// ---- Devices/Basic/FB_DeviceReal.TcPOU
(*
	Basic device with extended interface:
	nControl BYTE: From TwinCAT >>> To Unity
	nStatus BYTE: FROM Unity >>> TO TwinCAT	
	fControlData REAL: From TwinCAT >>> To Unity
	fStatusData REAL: FROM Unity >>> TO TwinCAT	
*)
FUNCTION_BLOCK FB_DeviceReal EXTENDS FB_LinkDataReal
VAR_INPUT		
	nControl  			: BYTE;
	fControlData  		: REAL;
END_VAR

VAR_OUTPUT
	nStatus  			: BYTE;
	fStatusData  		: REAL;
END_VAR

SUPER^();
Control := nControl;
ControlData := fControlData;
nStatus := Status;
fStatusData := StatusData;

END_FUNCTION_BLOCK

// ---- Common/Links/FB_LinkDataReal.TcPOU
(*
	Link component with additional interface:
	Control BYTE: From TwinCAT >>> To Unity	(Default)
	Status BYTE: FROM Unity >>> TO TwinCAT	(Default)
	ControlData REAL: From TwinCAT >>> To Unity		
	StatusData REAL: FROM Unity >>> TO TwinCAT		
*)
FUNCTION_BLOCK FB_LinkDataReal EXTENDS FB_LinkDevice
VAR	
	{attribute 'simulation_interface'}
	ControlData			AT %Q* : REAL;
	{attribute 'simulation_interface'}
	StatusData			AT %I* : REAL;
END_VAR

SUPER^();

METHOD INTERNAL GetLinkControlData : REAL
GetLinkControlData := ControlData;
END_METHOD

METHOD INTERNAL SetLinkStatusData : BOOL
VAR_INPUT
	fStatusData : REAL;
END_VAR
StatusData := fStatusData;
END_METHOD

END_FUNCTION_BLOCK

// ---- Tests/Devices/FB_Drive_Test.TcPOU
FUNCTION_BLOCK FB_Drive_Test EXTENDS TcUnit.FB_TestSuite
VAR
	_fbDrive 			: FB_Drive;
	_nExpectedByte 		: BYTE;
	_nResultByte 		: BYTE;
	_fExpectedReal 		: REAL;
	_fResultReal 		: REAL;
END_VAR

TEST('Set nControl');
_nExpectedByte := 255;
_fbDrive.nControl := _nExpectedByte;
_fbDrive();
_nResultByte := _fbDrive.GetControl();

AssertEquals(Expected := _nExpectedByte,
             Actual := _nResultByte,
             Message := 'Value is not correct');	
TEST_FINISHED();

TEST('Get nStatus');
_nExpectedByte := 255;
_fbDrive.SetStatus(_nExpectedByte);
_fbDrive();
_nResultByte := _fbDrive.nStatus;

AssertEquals(Expected := _nExpectedByte,
             Actual := _nResultByte,
             Message := 'Value is not correct');	
TEST_FINISHED();

TEST('Set fTargetValue_1');
_fExpectedReal := 1000;
_fbDrive.fTargetValue := _fExpectedReal;
_fbDrive();
_fResultReal := _fbDrive.GetLinkControlData();

AssertEquals(Expected := _fExpectedReal,
             Actual := _fResultReal,
             Message := 'Value is not correct');	
TEST_FINISHED();

TEST('Set fTargetValue_2');
_fExpectedReal := -1000;
_fbDrive.fTargetValue := _fExpectedReal;
_fbDrive();
_fResultReal := _fbDrive.GetLinkControlData();

AssertEquals(Expected := _fExpectedReal,
             Actual := _fResultReal,
             Message := 'Value is not correct');	
TEST_FINISHED();

TEST('Get fActualValue_1');
_fExpectedReal := 1000;
_fbDrive.SetLinkStatusData(_fExpectedReal);
_fbDrive();
_fResultReal := _fbDrive.fActualValue;

AssertEquals(Expected := _fExpectedReal,
             Actual := _fResultReal,
             Message := 'Value is not correct');	
TEST_FINISHED();

TEST('Get fActualValue_2');
_fExpectedReal := -1000;
_fbDrive.SetLinkStatusData(_fExpectedReal);
_fbDrive();
_fResultReal := _fbDrive.fActualValue;

AssertEquals(Expected := _fExpectedReal,
             Actual := _fResultReal,
             Message := 'Value is not correct');	
TEST_FINISHED();

END_FUNCTION_BLOCK

// ---- Devices/Basic/FB_Drive.TcPOU
(*
	Basic drive interface:
	nControl BYTE: From TwinCAT >>> To Unity
	nStatus BYTE: FROM Unity >>> TO TwinCAT	
	fTargetValue REAL: From TwinCAT >>> To Unity
	fActualValue REAL: FROM Unity >>> TO TwinCAT	
*)
FUNCTION_BLOCK FB_Drive EXTENDS FB_LinkDataREAL
VAR_INPUT
	nControl  		: BYTE;
	fTargetValue 	: REAL; //Target value to drive
END_VAR

VAR_OUTPUT
	nStatus  		: BYTE;
	fActualValue 	: REAL; //Actual value from drive
END_VAR

SUPER^();
Control := nControl;
ControlData := fTargetValue;
nStatus := Status;
fActualValue := StatusData;

END_FUNCTION_BLOCK

// ---- Tests/Devices/FB_Lamp_Test.TcPOU
FUNCTION_BLOCK FB_Lamp_Test EXTENDS TcUnit.FB_TestSuite
VAR
	_fbLamp : FB_Lamp;
	_nExpected : BYTE;
	_nResult : BYTE;
	_bExpected : BOOL;
	_bResult : BOOL;
END_VAR

TEST('Set bEnable TRUE');			 
_fbLamp.bEnable := TRUE; 
_fbLamp();
_nExpected := 1;
_nResult := _fbLamp.GetControl();
AssertEquals(Expected := _nExpected,
             Actual := _nResult,
             Message := 'Control value is not correct');	 
TEST_FINISHED();

TEST('Set bEnable FALSE');			 
_fbLamp.bEnable := FALSE; 
_fbLamp();
_nExpected := 0;
_nResult := _fbLamp.GetControl();
AssertEquals(Expected := _nExpected,
             Actual := _nResult,
             Message := 'Control value is not correct');	 
TEST_FINISHED();

END_FUNCTION_BLOCK

// ---- Devices/Basic/FB_Lamp.TcPOU
(*
	Default Lamp device
*)
FUNCTION_BLOCK FB_Lamp EXTENDS FB_LinkDevice 
VAR_INPUT
	bEnable		: BOOL; //0-Lamp OFF, 1 - Lamp ON
END_VAR

SUPER^();
Control.0 := bEnable;

END_FUNCTION_BLOCK

// ---- Tests/Devices/FB_Reader_Test.TcPOU
FUNCTION_BLOCK FB_Reader_Test EXTENDS TcUnit.FB_TestSuite
VAR
	_fbDevice 		: FB_Reader;
	_nExpected 		: LWORD;
	_nResult 		: LWORD;
	_nValue 		: LWORD := 16#FFAABBCC;
END_VAR

TEST('Set nControl');
_nExpected := 255;
_fbDevice.nControl := 255;
_fbDevice();
_nResult := _fbDevice.GetControl();

AssertEquals(Expected := _nExpected,
             Actual := _nResult,
             Message := 'Value is not correct');	
TEST_FINISHED();

TEST('Set nCommand');
_nExpected := _nValue;
_fbDevice.nCommand := _nExpected;
_fbDevice();
_nResult := _fbDevice.GetLinkControlData();

AssertEquals(Expected := _nExpected,
             Actual := _nResult,
             Message := 'Value is not correct');	
TEST_FINISHED();

TEST('Get nStatus');
_nExpected := 255;
_fbDevice.SetStatus(255);
_fbDevice();
_nResult := _fbDevice.nStatus;

AssertEquals(Expected := _nExpected,
             Actual := _nResult,
             Message := 'Value is not correct');	
TEST_FINISHED();

TEST('Get nResult');
_nExpected := _nValue;
_fbDevice.SetLinkStatusData(_nExpected);
_fbDevice();
_nResult := _fbDevice.nResult;

AssertEquals(Expected := _nExpected,
             Actual := _nResult,
             Message := 'Value is not correct');	
TEST_FINISHED();

END_FUNCTION_BLOCK

// ---- Devices/Basic/FB_Reader.TcPOU
(*
	Default reader device	
*)
FUNCTION_BLOCK FB_Reader EXTENDS FB_LinkDataLWORD
VAR_INPUT
	nControl  		: BYTE;
	nCommand 		: ULINT; //Command ID
END_VAR

VAR_OUTPUT
	nStatus  		: BYTE;
	nResult			: ULINT; //Result Data
END_VAR

SUPER^();
Control := nControl;
ControlData := ULINT_TO_LWORD(nCommand);
nStatus := Status;
nResult := LWORD_TO_ULINT(StatusData);

END_FUNCTION_BLOCK

// ---- Tests/Devices/FB_SensorAnalog_Test.TcPOU
FUNCTION_BLOCK FB_SensorAnalog_Test EXTENDS TcUnit.FB_TestSuite
VAR
	_fbSensorAnalog 	: FB_SensorAnalog;
	_nExpectedByte 		: BYTE;
	_nResultByte 		: BYTE;
	_nExpectedUInt 		: UINT;
	_nResultUInt 		: UINT;
	_fExpectedReal 		: REAL;
	_fResultReal 		: REAL;
END_VAR

TEST('Set nControl');
_nExpectedByte := 255;
_fbSensorAnalog.nControl := _nExpectedByte;
_fbSensorAnalog();
_nResultByte := _fbSensorAnalog.GetControl();

AssertEquals(Expected := _nExpectedByte,
             Actual := _nResultByte,
             Message := 'Value is not correct');	
TEST_FINISHED();

TEST('Get nStatus');
_nExpectedByte := 255;
_fbSensorAnalog.SetStatus(_nExpectedByte);
_fbSensorAnalog();
_nResultByte := _fbSensorAnalog.nStatus;

AssertEquals(Expected := _nExpectedByte,
             Actual := _nResultByte,
             Message := 'Value is not correct');	
TEST_FINISHED();


TEST('Get fValue');
_fExpectedReal := 50;
_nExpectedUInt := 16#8000;
_fbSensorAnalog.SetLinkStatusData(_fExpectedReal);
_fbSensorAnalog();
_fResultReal := _fbSensorAnalog.fValue;
_nResultUInt := _fbSensorAnalog.nValue;

AssertEquals(Expected := _fExpectedReal,
             Actual := _fResultReal,
             Message := 'fValue is not correct');	
AssertEquals(Expected := _nExpectedUInt,
             Actual := _nResultUInt,
             Message := 'nValue is not correct');
TEST_FINISHED();

END_FUNCTION_BLOCK

// ---- Devices/Basic/FB_SensorAnalog.TcPOU
(*
	Default analog sensor device. 
	The stConfig structure is used to configure the scaling factor for transforming values into real-world units.
*)
FUNCTION_BLOCK FB_SensorAnalog EXTENDS FB_LinkDataReal 
VAR_INPUT
	nControl  		: BYTE;
	stConfig		: ST_ScaleConfig;
END_VAR

VAR_OUTPUT	
	nStatus  		: BYTE;
	nValue			: UINT;
	fValue			: REAL;
END_VAR

SUPER^();
Control := nControl;
fValue := StatusData;
nValue := LREAL_TO_UINT(F_ScaleLREAL(fValue, stConfig.fInputMin, stConfig.fInputMax, stConfig.fOutputMin, stConfig.fOutputMax));
nStatus := Status;

END_FUNCTION_BLOCK

// ---- Tests/Devices/FB_SensorBinary_Test.TcPOU
FUNCTION_BLOCK FB_SensorBinary_Test EXTENDS TcUnit.FB_TestSuite
VAR
	_fbSensorBinary 	: FB_SensorBinary;
	_nExpected 			: BYTE;
	_nResult 			: BYTE;
	_bExpected 			: BOOL;
	_bResult 			: BOOL;
END_VAR

TEST('Get bValue FALSE');
_fbSensorBinary.SetStatus(0);
_fbSensorBinary();
_bExpected := FALSE;
_bResult := _fbSensorBinary.bValue;

AssertEquals(Expected := _bExpected,
             Actual := _bResult,
             Message := 'Value is not correct');	
TEST_FINISHED();

TEST('Get bValue TRUE');	
_fbSensorBinary.SetStatus(1);
_fbSensorBinary();
_bExpected := 1;
_bResult := _fbSensorBinary.bValue;
AssertEquals(Expected := _bExpected,
             Actual := _bResult,
             Message := 'Control value is not correct');	 
TEST_FINISHED();

END_FUNCTION_BLOCK

// ---- Devices/Basic/FB_SensorBinary.TcPOU
(*
	Default binary sensor device.
*)
FUNCTION_BLOCK FB_SensorBinary EXTENDS FB_LinkDevice 
VAR_OUTPUT
	bValue		: BOOL; 
END_VAR

SUPER^();
bValue := Status.0;

END_FUNCTION_BLOCK

// ---- Tests/Devices/FB_Robot_Test.TcPOU
FUNCTION_BLOCK FB_Robot_Test EXTENDS TcUnit.FB_TestSuite
VAR
	_fbRobot 			: FB_Robot;
	_nExpectedByte 		: BYTE;
	_nResultByte 		: BYTE;
	_aExpectedJoints 	: ARRAY[0..11] OF REAL := [11, 22, 33, 44, 55, 66, 77, 88, 99, 1010, 1111, 1212];	
	_aResultJoints 		: ARRAY[0..11] OF REAL;	
	_nJointCount 		: INT := 12;
END_VAR

TEST('Set nControl');
_nExpectedByte := 255;
_fbRobot.nControl := _nExpectedByte;
_fbRobot();
_nResultByte := _fbRobot.GetControl();

AssertEquals(Expected := _nExpectedByte,
             Actual := _nResultByte,
             Message := 'Value is not correct');	
TEST_FINISHED();

TEST('Get nStatus');
_nExpectedByte := 255;
_fbRobot.SetStatus(_nExpectedByte);
_fbRobot();
_nResultByte := _fbRobot.nStatus;

AssertEquals(Expected := _nExpectedByte,
             Actual := _nResultByte,
             Message := 'Value is not correct');	
TEST_FINISHED();

TestSetJoint('Set Joint 1', 0, 100);
TestSetJoint('Set Joint 2', 1, 100);
TestSetJoint('Set Joint 3', 2, 100);
TestSetJoint('Set Joint 4', 3, 100);
TestSetJoint('Set Joint 5', 4, 100);
TestSetJoint('Set Joint 6', 5, 100);
TestSetJoint('Set Joint EXT1', 6, 100);
TestSetJoint('Set Joint EXT2', 7, 100);
TestSetJoint('Set Joint EXT3', 8, 100);
TestSetJoint('Set Joint EXT4', 9, 100);
TestSetJoint('Set Joint EXT5', 10, 100);
TestSetJoint('Set Joint EXT6', 11, 100);

TestGetJoint('Get Joint 1', 0, 100);
TestGetJoint('Get Joint 2', 1, 100);
TestGetJoint('Get Joint 3', 2, 100);
TestGetJoint('Get Joint 4', 3, 100);
TestGetJoint('Get Joint 5', 4, 100);
TestGetJoint('Get Joint 6', 5, 100);
TestGetJoint('Get Joint EXT1', 6, 100);
TestGetJoint('Get Joint EXT2', 7, 100);
TestGetJoint('Get Joint EXT3', 8, 100);
TestGetJoint('Get Joint EXT4', 9, 100);
TestGetJoint('Get Joint EXT5', 10, 100);
TestGetJoint('Get Joint EXT6', 11, 100);

TEST('Set Joints wia Pointer');
_fbRobot.ConnectJoints(_aExpectedJoints, 12);
_fbRobot();
_aResultJoints := _fbRobot.GetJointsTarget();
AssertEquals(Expected := _aExpectedJoints,
             Actual := _aResultJoints,
             Message := 'Value is not correct');	
TEST_FINISHED();

METHOD TestGetJoint : BOOL
VAR_INPUT
	sName : T_MaxString;
	nJointIndex : INT;
	fValue : REAL;
END_VAR

VAR
	fbRobot : FB_Robot;	
	fResult : REAL;		
	aExpectedJoints : ARRAY[0..11] OF REAL;
END_VAR
TEST(sName);

aExpectedJoints[nJointIndex] := fValue;
fbRobot.SetJointsStatus(aExpectedJoints);
fbRobot();
fResult := fbRobot.aJointStatus[nJointIndex];

AssertEquals(Expected := fValue,
             Actual := fResult,
             Message := 'Result value is not correct');	
	 
TEST_FINISHED();
END_METHOD

METHOD TestSetJoint : BOOL
VAR_INPUT
	sName : T_MaxString;
	nJointIndex : INT;
	fValue : REAL;
END_VAR

VAR
	fbRobot : FB_Robot;	
	fResult : REAL;		
	aResultJoints : ARRAY[0..11] OF REAL;
END_VAR
TEST(sName);

fbRobot.aJointTarget[nJointIndex] := fValue;
fbRobot();
aResultJoints := fbRobot.GetJointsTarget();
fResult := aResultJoints[nJointIndex];

AssertEquals(Expected := fValue,
             Actual := fResult,
             Message := 'Result value is not correct');	
	 
TEST_FINISHED();
END_METHOD

END_FUNCTION_BLOCK

// ---- Devices/Basic/FB_Robot.TcPOU
(*
	Default robot component with 12 axis interface	
*)
FUNCTION_BLOCK FB_Robot EXTENDS FB_LinkDevice
VAR_INPUT
	nControl  			: BYTE;	
	aJointTarget 		: ARRAY[0..11] OF REAL;	
END_VAR

VAR_OUTPUT
	nStatus  			: BYTE;
	aJointStatus 		: ARRAY[0..11] OF REAL;
END_VAR

VAR
	{attribute 'simulation_interface'}
	JointStatus AT %I* 	: ARRAY[0..11] OF REAL;
	{attribute 'simulation_interface'}
	JointTarget AT %Q* 	: ARRAY[0..11] OF REAL;
	
	{attribute 'hide'}
	_adrData			: LWORD;
	{attribute 'hide'}
	_nDataLength 		: UDINT;	
END_VAR

SUPER^();

IF (_adrData <> 0) THEN	
	MEMCPY(ADR(aJointTarget), _adrData, _nDataLength);
END_IF

Control := nControl;
MEMCPY(ADR(JointTarget), ADR(aJointTarget), 12 * 4);
MEMCPY(ADR(aJointStatus), ADR(JointStatus), 12 * 4);
nStatus := Status;

(*
	Assign the joint memory area for cyclic data exchange
*)
METHOD ConnectJoints : BOOL
VAR_INPUT
	Joints : ANY; //Adress to joints memmory area
	nJointCount : UDINT; //Number of joints
END_VAR
_adrData := Joints.pValue;
_nDataLength := LIMIT(0, nJointCount * 4, 12 * 4);
END_METHOD

METHOD INTERNAL GetJointsTarget : ARRAY[0..11] OF REAL;
GetJointsTarget := JointTarget;
END_METHOD

METHOD INTERNAL SetJointsStatus : BOOL
VAR_INPUT
	aJointsStatus : ARRAY[0..11] OF REAL;
END_VAR
JointStatus := aJointsStatus;
END_METHOD

END_FUNCTION_BLOCK

// ---- Tests/Common/FB_AdsMessageHandler_Test.TcPOU
FUNCTION_BLOCK FB_AdsMessageHandler_Test EXTENDS TcUnit.FB_TestSuite
VAR
	_stAdsMessageSend 		: ST_AdsMessage;
END_VAR

_stAdsMessageSend.nIdxGrp := 16#80000005;
_stAdsMessageSend.nIdxOffs := 7;
TestCaseWrite('ADS Write Indication 1', _stAdsMessageSend);

_stAdsMessageSend.nIdxGrp := 16#80000006;
_stAdsMessageSend.nIdxOffs := 8;
TestCaseWrite('ADS Write Indication 2', _stAdsMessageSend);

_stAdsMessageSend.nIdxGrp := 16#80000007;
_stAdsMessageSend.nIdxOffs := 9;
TestCaseWrite('ADS Write Indication 3', _stAdsMessageSend);

_stAdsMessageSend.nIdxGrp := 16#80000005;
_stAdsMessageSend.nIdxOffs := 7;
TestCaseRead('ADS Read Indication 1', _stAdsMessageSend);

_stAdsMessageSend.nIdxGrp := 16#80000006;
_stAdsMessageSend.nIdxOffs := 8;
TestCaseRead('ADS Read Indication 2', _stAdsMessageSend);

_stAdsMessageSend.nIdxGrp := 16#80000007;
_stAdsMessageSend.nIdxOffs := 9;
TestCaseRead('ADS Read Indication 3', _stAdsMessageSend);

METHOD TestCaseRead : REFERENCE TO FB_Test
VAR_INPUT
	sName 					: T_MaxString;
	stAdsMessage 			: ST_AdsMessage;
END_VAR

VAR
	fbAdsMessageHandler 	: FB_AdsMessageHandler;		
	fbAdsRead				: ADSREAD := (NETID := '', PORT := 851, TMOUT := DEFAULT_ADS_TIMEOUT);
	aData 					: ARRAY[0..5] OF BYTE;
	bResult 				: BOOL; 	
	stAdsMessageResult 		: ST_AdsMessage;
END_VAR
TEST(sName);

fbAdsRead(READ := FALSE);
fbAdsRead(IDXGRP := _stAdsMessageSend.nIdxGrp, 
		IDXOFFS := _stAdsMessageSend.nIdxOffs, 
        LEN := _stAdsMessageSend.nLength, 
		DESTADDR := ADR(aData), 
        READ := TRUE);			

fbAdsMessageHandler.bVerbose := TRUE;			
fbAdsMessageHandler();

bResult := fbAdsMessageHandler.bIsAdsMessageReadValid;
stAdsMessageResult := fbAdsMessageHandler.stAdsMessageRead;

AssertTrue(bResult, 'Result value is not correct');

AssertEquals(Expected := stAdsMessage.tNetID,
Actual := stAdsMessageResult.tNetID,
Message := 'tNetID is not valid');

AssertEquals(Expected := stAdsMessage.nIdxGrp,
Actual := stAdsMessageResult.nIdxGrp,
Message := 'nIdxGrp is not valid');

AssertEquals(Expected := stAdsMessage.nIdxOffs,
Actual := stAdsMessageResult.nIdxOffs,
Message := 'nIdxOffs is not valid');

AssertEquals(Expected := stAdsMessage.nLength,
Actual := stAdsMessageResult.nLength,
Message := 'nLength is not valid');

TEST_FINISHED();
END_METHOD

METHOD TestCaseWrite : REFERENCE TO FB_Test
VAR_INPUT
	sName 					: T_MaxString;
	stAdsMessage 			: ST_AdsMessage;
END_VAR

VAR
	fbAdsMessageHandler 	: FB_AdsMessageHandler;		
	fbAdsWrite				: ADSWRITE := (NETID := '', PORT := 851, TMOUT := DEFAULT_ADS_TIMEOUT);
	aData 					: ARRAY[0..5] OF BYTE;
	bResult 				: BOOL; 	
	stAdsMessageResult 		: ST_AdsMessage;
END_VAR
TEST(sName);

fbAdsWrite(WRITE := FALSE);
fbAdsWrite(	IDXGRP := _stAdsMessageSend.nIdxGrp, 
			IDXOFFS := _stAdsMessageSend.nIdxOffs, 
            LEN := _stAdsMessageSend.nLength, 
			SRCADDR := ADR(aData), 
            WRITE := TRUE);			

fbAdsMessageHandler.bVerbose := TRUE;			
fbAdsMessageHandler();

bResult := fbAdsMessageHandler.bIsAdsMessageWriteValid;
stAdsMessageResult := fbAdsMessageHandler.stAdsMessageWrite;

AssertTrue(bResult, 'Result value is not correct');

AssertEquals(Expected := stAdsMessage.tNetID,
Actual := stAdsMessageResult.tNetID,
Message := 'tNetID is not valid');

AssertEquals(Expected := stAdsMessage.nIdxGrp,
Actual := stAdsMessageResult.nIdxGrp,
Message := 'nIdxGrp is not valid');

AssertEquals(Expected := stAdsMessage.nIdxOffs,
Actual := stAdsMessageResult.nIdxOffs,
Message := 'nIdxOffs is not valid');

AssertEquals(Expected := stAdsMessage.nLength,
Actual := stAdsMessageResult.nLength,
Message := 'nLength is not valid');

TEST_FINISHED();
END_METHOD

END_FUNCTION_BLOCK

// ---- Tests/Common/FB_RecordData_Test.TcPOU
FUNCTION_BLOCK FB_RecordData_Test EXTENDS TcUnit.FB_TestSuite
VAR
	_fbAdsMessageHandler 	: FB_AdsMessageHandler;
	_fbRecordData 			: FB_RecordData(refAdsMessageHandler := _fbAdsMessageHandler);		
	_stAdsHandlerMessage 	: ST_AdsMessage;
	_stDeviceMessage 		: ST_AdsMessage;
END_VAR

TestCasesCompare();
TestGetReadIndication();
TestGetWriteIndication();
TestSendReadResponse();
TestSendWriteResponse();
TestAutoResponseWriteMessage();
TestAutoResponseReadMessage();

METHOD TestAutoResponseReadMessage : REFERENCE TO FB_Test
VAR
	fbAdsRead				: ADSREAD := (NETID := '', PORT := 851, TMOUT := DEFAULT_ADS_TIMEOUT);
	stAdsMessage			: REFERENCE TO ST_AdsMessage;
	nData					: BYTE;
	bResult 				: BOOL;
	bResultPort 			: T_AmsPort;
	nExpectedPort			: T_AmsPort;
END_VAR
TEST('Auto Response Ads Read Message');

_stAdsHandlerMessage.tPort := 351; 
_stAdsHandlerMessage.nInvokeID := 500;
_stAdsHandlerMessage.nIdxGrp := 16#80000001;
_stAdsHandlerMessage.nIdxOffs := 10;
_stDeviceMessage.tPort := 351;
_stDeviceMessage.nInvokeID := 500;
_stDeviceMessage.nIdxGrp := 16#80000001;
_stDeviceMessage.nIdxOffs := 10;

fbAdsRead(READ := FALSE);
fbAdsRead(	IDXGRP := _stAdsHandlerMessage.nIdxGrp, 
			IDXOFFS := _stAdsHandlerMessage.nIdxOffs, 
        	LEN := _stAdsHandlerMessage.nLength, 
			DESTADDR := ADR(nData), 
        	READ := TRUE);			

_fbAdsMessageHandler.bLog := TRUE;
_fbAdsMessageHandler.bVerbose := TRUE;	
_fbRecordData.eControllerType := E_ControllerType.PlcSimAdvanced;

_fbRecordData();		
_fbAdsMessageHandler();

bResult := _fbAdsMessageHandler.bIsAdsMessageReadValid;
AssertTrue(bResult, 'AdsMessageReadValid expected TRUE');

_fbRecordData();	
_fbAdsMessageHandler();
bResult := _fbAdsMessageHandler.bIsAdsMessageReadValid;
AssertFalse(bResult, 'AdsMessageReadValid expected FALSE');

nExpectedPort := 0;
bResultPort := _fbAdsMessageHandler.stAdsMessageRead.tPort;

AssertEquals(Expected := nExpectedPort,
	Actual := bResultPort,
	Message := 'tPort value is incorrect');

TEST_FINISHED();
END_METHOD

METHOD TestAutoResponseWriteMessage : REFERENCE TO FB_Test
VAR
	fbAdsWrite				: ADSWRITE := (NETID := '', PORT := 851, TMOUT := DEFAULT_ADS_TIMEOUT);
	stAdsMessage			: REFERENCE TO ST_AdsMessage;
	nData					: BYTE;
	bResult 				: BOOL;
	bResultPort 			: T_AmsPort;
	nExpectedPort			: T_AmsPort;
END_VAR
TEST('Auto Response Ads Write Message');

_stAdsHandlerMessage.tPort := 351; 
_stAdsHandlerMessage.nInvokeID := 500;
_stAdsHandlerMessage.nIdxGrp := 16#80000001;
_stAdsHandlerMessage.nIdxOffs := 10;
_stDeviceMessage.tPort := 351;
_stDeviceMessage.nInvokeID := 500;
_stDeviceMessage.nIdxGrp := 16#80000001;
_stDeviceMessage.nIdxOffs := 10;

fbAdsWrite(WRITE := FALSE);
fbAdsWrite(	IDXGRP := _stAdsHandlerMessage.nIdxGrp, 
			IDXOFFS := _stAdsHandlerMessage.nIdxOffs, 
           	LEN := _stAdsHandlerMessage.nLength, 
			SRCADDR := ADR(nData), 
           	WRITE := TRUE);			

_fbAdsMessageHandler.bLog := TRUE;
_fbAdsMessageHandler.bVerbose := TRUE;	
_fbRecordData.eControllerType := E_ControllerType.PlcSimAdvanced;

_fbRecordData();		
_fbAdsMessageHandler();

bResult := _fbAdsMessageHandler.bIsAdsMessageWriteValid;
AssertTrue(bResult, 'AdsMessageWriteValid expected TRUE');

_fbRecordData();	
_fbAdsMessageHandler();
bResult := _fbAdsMessageHandler.bIsAdsMessageWriteValid;
AssertFalse(bResult, 'AdsMessageWriteValid expected FALSE');

nExpectedPort := 0;
bResultPort := _fbAdsMessageHandler.stAdsMessageWrite.tPort;

AssertEquals(Expected := nExpectedPort,
	Actual := bResultPort,
	Message := 'tPort value is incorrect');

TEST_FINISHED();
END_METHOD

METHOD TestCaseCompare : REFERENCE TO FB_Test
VAR_INPUT
	sName 					: T_MaxString;
	stAdsHandlerMessage 	: ST_AdsMessage;
	stDeviceMessage 		: ST_AdsMessage;
	bExpected				: BOOL;
END_VAR

VAR
	bResult 				: BOOL;
END_VAR
TEST(sName);

bResult := _fbRecordData.DataValid(stDeviceMessage, stAdsHandlerMessage);

AssertEquals(Expected := bExpected,
	Actual := bResult,
	Message := 'Expected compare result is wrong');

IF bResult AND bExpected THEN
	bResult := stAdsHandlerMessage.tPort = 0;
	AssertTrue(bResult, 'tPort must be 0');
END_IF
	
	
TEST_FINISHED();
END_METHOD

ACTION TestCasesCompare:
(*Test ADS Message compare*)
_stAdsHandlerMessage.tPort := 351; 
_stAdsHandlerMessage.nInvokeID := 500;
_stAdsHandlerMessage.nIdxGrp := 16#80000001;
_stAdsHandlerMessage.nIdxOffs := 10;
_stDeviceMessage.tPort := 351;
_stDeviceMessage.nInvokeID := 500;
_stDeviceMessage.nIdxGrp := 16#80000001;
_stDeviceMessage.nIdxOffs := 10;
TestCaseCompare('Compare TRUE 1', _stAdsHandlerMessage, _stDeviceMessage, TRUE);

_stAdsHandlerMessage.tPort := 351; 
_stAdsHandlerMessage.nInvokeID := 16#12340011;
_stAdsHandlerMessage.nIdxGrp := 16#80000001;
_stAdsHandlerMessage.nIdxOffs := 10;
_stDeviceMessage.tPort := 351;
_stDeviceMessage.nInvokeID := 16#43210011;
_stDeviceMessage.nIdxGrp := 16#80000001;
_stDeviceMessage.nIdxOffs := 10;
TestCaseCompare('Compare TRUE - InvokeID', _stAdsHandlerMessage, _stDeviceMessage, TRUE);

_stAdsHandlerMessage.tPort := 351; 
_stAdsHandlerMessage.nInvokeID := 16#12340011;
_stAdsHandlerMessage.nIdxGrp := 16#80000001;
_stAdsHandlerMessage.nIdxOffs := 10;
_stDeviceMessage.tPort := 351;
_stDeviceMessage.nInvokeID := 16#43210011;
_stDeviceMessage.nIdxGrp := 16#80000001;
_stDeviceMessage.nIdxOffs := 10;
TestCaseCompare('Compare TRUE - nIdxOffs', _stAdsHandlerMessage, _stDeviceMessage, TRUE);

_stAdsHandlerMessage.tPort := 351; 
_stAdsHandlerMessage.nInvokeID := 16#12340011;
_stAdsHandlerMessage.nIdxGrp := 16#80000001;
_stAdsHandlerMessage.nIdxOffs := 10;
_stDeviceMessage.tPort := 351;
_stDeviceMessage.nInvokeID := 16#43210011;
_stDeviceMessage.nIdxGrp := 16#80000001;
_stDeviceMessage.nIdxOffs := 16#FFFFFFFF;
TestCaseCompare('Compare TRUE - nIdxOffs 16#FFFFFFFF', _stAdsHandlerMessage, _stDeviceMessage, TRUE);

_stAdsHandlerMessage.tPort := 351; 
_stAdsHandlerMessage.nInvokeID := 16#12340011;
_stAdsHandlerMessage.nIdxGrp := 16#12340011;
_stAdsHandlerMessage.nIdxOffs := 10;
_stDeviceMessage.tPort := 351;
_stDeviceMessage.nInvokeID := 16#43210011;
_stDeviceMessage.nIdxGrp := 16#43210011;
_stDeviceMessage.nIdxOffs := 10;
TestCaseCompare('Compare TRUE - nIdxGrp', _stAdsHandlerMessage, _stDeviceMessage, TRUE);

_stAdsHandlerMessage.tPort := 351; 
_stAdsHandlerMessage.nInvokeID := 16#12340011;
_stAdsHandlerMessage.nIdxGrp := 16#12340011;
_stAdsHandlerMessage.nIdxOffs := 10;
_stDeviceMessage.tPort := 351;
_stDeviceMessage.nInvokeID := 16#43210011;
_stDeviceMessage.nIdxGrp := 0;
_stDeviceMessage.nIdxOffs := 10;
TestCaseCompare('Compare TRUE - nIdxGrp 0', _stAdsHandlerMessage, _stDeviceMessage, TRUE);

_stAdsHandlerMessage.tPort := 0; 
_stAdsHandlerMessage.nInvokeID := 500;
_stAdsHandlerMessage.nIdxGrp := 16#80000001;
_stAdsHandlerMessage.nIdxOffs := 10;
_stDeviceMessage.tPort := 351;
_stDeviceMessage.nInvokeID := 500;
_stDeviceMessage.nIdxGrp := 16#80000001;
_stDeviceMessage.nIdxOffs := 10;
TestCaseCompare('Compare FALSE - AdsHandler Port 0', _stAdsHandlerMessage, _stDeviceMessage, FALSE);

_stAdsHandlerMessage.tPort := 351; 
_stAdsHandlerMessage.nInvokeID := 16#12340010;
_stAdsHandlerMessage.nIdxGrp := 16#80000001;
_stAdsHandlerMessage.nIdxOffs := 10;
_stDeviceMessage.tPort := 351;
_stDeviceMessage.nInvokeID := 16#43210001;
_stDeviceMessage.nIdxGrp := 16#80000001;
_stDeviceMessage.nIdxOffs := 10;
TestCaseCompare('Compare FALSE - InvokeID', _stAdsHandlerMessage, _stDeviceMessage, FALSE);

_stAdsHandlerMessage.tPort := 351; 
_stAdsHandlerMessage.nInvokeID := 16#12340011;
_stAdsHandlerMessage.nIdxGrp := 16#12340000;
_stAdsHandlerMessage.nIdxOffs := 10;
_stDeviceMessage.tPort := 351;
_stDeviceMessage.nInvokeID := 16#43210000;
_stDeviceMessage.nIdxGrp := 16#43210022;
_stDeviceMessage.nIdxOffs := 10;
TestCaseCompare('Compare FALSE - nIdxGrp', _stAdsHandlerMessage, _stDeviceMessage, FALSE);

_stAdsHandlerMessage.tPort := 351; 
_stAdsHandlerMessage.nInvokeID := 16#12340011;
_stAdsHandlerMessage.nIdxGrp := 16#12340000;
_stAdsHandlerMessage.nIdxOffs := 20;
_stDeviceMessage.tPort := 351;
_stDeviceMessage.nInvokeID := 16#43210000;
_stDeviceMessage.nIdxGrp := 16#43210000;
_stDeviceMessage.nIdxOffs := 10;
TestCaseCompare('Compare FALSE - nIdxOffs', _stAdsHandlerMessage, _stDeviceMessage, FALSE);
END_ACTION

METHOD TestGetReadIndication : REFERENCE TO FB_Test
VAR	
	fbAdsRead				: ADSREAD := (NETID := '', PORT := 851, TMOUT := DEFAULT_ADS_TIMEOUT);
	stAdsMessage			: REFERENCE TO ST_AdsMessage;
	nData					: BYTE;
	bResult 				: BOOL;
END_VAR
TEST('Get Read Indication');

_stAdsHandlerMessage.tPort := 351; 
_stAdsHandlerMessage.nInvokeID := 500;
_stAdsHandlerMessage.nIdxGrp := 16#80000001;
_stAdsHandlerMessage.nIdxOffs := 10;
_stDeviceMessage.tPort := 351;
_stDeviceMessage.nInvokeID := 500;
_stDeviceMessage.nIdxGrp := 16#80000001;
_stDeviceMessage.nIdxOffs := 10;

fbAdsRead(READ := FALSE);
fbAdsRead(	IDXGRP := _stAdsHandlerMessage.nIdxGrp, 
			IDXOFFS := _stAdsHandlerMessage.nIdxOffs, 
        	LEN := _stAdsHandlerMessage.nLength, 
			DESTADDR := ADR(nData), 
        	READ := TRUE);			

_fbAdsMessageHandler.bLog := TRUE;
_fbAdsMessageHandler.bVerbose := TRUE;			
_fbAdsMessageHandler();

_fbRecordData.eControllerType := E_ControllerType.PlcSimAdvanced;

bResult := _fbRecordData.GetReadIndication(_stDeviceMessage);
stAdsMessage REF= _fbAdsMessageHandler.stAdsMessageRead;

AssertTrue(bResult, 'Result value is not correct');

bResult := stAdsMessage.tPort = 0;
AssertTrue(bResult, 'tPort must be 0');

TEST_FINISHED();
END_METHOD

METHOD TestGetWriteIndication : REFERENCE TO FB_Test
VAR	
	fbAdsWrite				: ADSWRITE := (NETID := '', PORT := 851, TMOUT := DEFAULT_ADS_TIMEOUT);
	stAdsMessage			: REFERENCE TO ST_AdsMessage;
	nData					: BYTE;
	bResult 				: BOOL;
END_VAR
TEST('Get Write Indication');

_stAdsHandlerMessage.tPort := 351; 
_stAdsHandlerMessage.nInvokeID := 500;
_stAdsHandlerMessage.nIdxGrp := 16#80000001;
_stAdsHandlerMessage.nIdxOffs := 10;
_stDeviceMessage.tPort := 351;
_stDeviceMessage.nInvokeID := 500;
_stDeviceMessage.nIdxGrp := 16#80000001;
_stDeviceMessage.nIdxOffs := 10;

fbAdsWrite(WRITE := FALSE);
fbAdsWrite(	IDXGRP := _stAdsHandlerMessage.nIdxGrp, 
			IDXOFFS := _stAdsHandlerMessage.nIdxOffs, 
           	LEN := _stAdsHandlerMessage.nLength, 
			SRCADDR := ADR(nData), 
           	WRITE := TRUE);			

_fbAdsMessageHandler.bLog := TRUE;
_fbAdsMessageHandler.bVerbose := TRUE;			
_fbAdsMessageHandler();

_fbRecordData.eControllerType := E_ControllerType.PlcSimAdvanced;

bResult := _fbRecordData.GetWriteIndication(_stDeviceMessage);
stAdsMessage REF= _fbAdsMessageHandler.stAdsMessageRead;

AssertTrue(bResult, 'Result value is not correct');

bResult := stAdsMessage.tPort = 0;
AssertTrue(bResult, 'tPort must be 0');

TEST_FINISHED();
END_METHOD

METHOD TestSendReadResponse : REFERENCE TO FB_Test
VAR
	stAdsMessage : ST_AdsMessage;
	hExpected : HRESULT;
	hRes : HRESULT;
END_VAR
TEST('Send Read Response');

stAdsMessage.tPort := 351;
stAdsMessage.nInvokeID := 500;
stAdsMessage.nIdxGrp := 16#80000001;
stAdsMessage.nIdxOffs := 10;

_fbAdsMessageHandler.bLog := TRUE;
_fbAdsMessageHandler.bVerbose := TRUE;			
_fbAdsMessageHandler();

_fbRecordData.eControllerType := E_ControllerType.PlcSimAdvanced;

hExpected := S_OK;
hRes := _fbRecordData.SendReadResponse(stAdsMessage);

AssertEquals(Expected := hExpected,
	Actual := hRes,
	Message := 'Expected result is not valid');
	
TEST_FINISHED();
END_METHOD

METHOD TestSendWriteResponse : REFERENCE TO FB_Test
VAR
	stAdsMessage : ST_AdsMessage;
	hExpected : HRESULT;
	hRes : HRESULT;
END_VAR
TEST('Send Write Response');

stAdsMessage.tPort := 351;
stAdsMessage.nInvokeID := 500;
stAdsMessage.nIdxGrp := 16#80000001;
stAdsMessage.nIdxOffs := 10;

_fbAdsMessageHandler.bLog := TRUE;
_fbAdsMessageHandler.bVerbose := TRUE;			
_fbAdsMessageHandler();

_fbRecordData.eControllerType := E_ControllerType.PlcSimAdvanced;

hExpected := S_OK;
hRes := _fbRecordData.SendReadResponse(stAdsMessage);

AssertEquals(Expected := hExpected,
	Actual := hRes,
	Message := 'Expected result is not valid');
	
TEST_FINISHED();
END_METHOD

END_FUNCTION_BLOCK

// ---- Tests/Common/FB_Encoder_Test.TcPOU
FUNCTION_BLOCK FB_Encoder_Test EXTENDS FB_TestSuite
VAR	
	_stConfig 				: ST_Encoder_Config;
	_fNumDen				: REAL;
	_fDenNum				: REAL;
END_VAR

_fNumDen := _stConfig.fNumerator / _stConfig.fDenominator;
_fDenNum := _stConfig.fDenominator / _stConfig.fNumerator;

TestCase_LREAL_TO_INC('LREAL_TO_INC 1', 0, 0, LREAL_TO_DINT(0*_fDenNum), _stConfig);
TestCase_LREAL_TO_INC('LREAL_TO_INC 2', 100, 1, LREAL_TO_DINT(100*_fDenNum), _stConfig);
TestCase_LREAL_TO_INC('LREAL_TO_INC 3', -100, 1, LREAL_TO_DINT(-100*_fDenNum), _stConfig);
TestCase_LREAL_TO_INC('LREAL_TO_INC 4', -100, -1, LREAL_TO_DINT(100*_fDenNum), _stConfig);

TestCase_INC_TO_LREAL('INC_TO_LREAL 1', LREAL_TO_DINT(0*_fDenNum), 0, 0, _stConfig);
TestCase_INC_TO_LREAL('INC_TO_LREAL 2', LREAL_TO_DINT(100*_fDenNum), 1, 100, _stConfig);
TestCase_INC_TO_LREAL('INC_TO_LREAL 3', -LREAL_TO_DINT(100*_fDenNum), 1, -100, _stConfig);
TestCase_INC_TO_LREAL('INC_TO_LREAL 4', -LREAL_TO_DINT(100*_fDenNum), -1, 100, _stConfig);

TestCaseEncoder('Absolute 1', 0, 0, LREAL_TO_DINT(0*_fDenNum), _stConfig);
TestCaseEncoder('Absolute 2', 100, 100, LREAL_TO_DINT(100*_fDenNum), _stConfig);
TestCaseEncoder('Absolute 3', -100, -100, LREAL_TO_DINT(-100*_fDenNum), _stConfig);

_stConfig.fGearFactor := -1;
TestCaseEncoder('Absolute with Factor 1', 0, 0, LREAL_TO_DINT(0*_fDenNum), _stConfig);
TestCaseEncoder('Absolute with Factor 2', 100, -100, LREAL_TO_DINT(-100*_fDenNum), _stConfig);
TestCaseEncoder('Absolute with Factor 3', -100, 100, LREAL_TO_DINT(100*_fDenNum), _stConfig);

_stConfig.fGearFactor := 1;
_stConfig.bInvertEncoderDirection := TRUE;
TestCaseEncoder('Absolute with Invert 1', 0, 0, LREAL_TO_DINT(0*_fDenNum), _stConfig);
TestCaseEncoder('Absolute with Invert 2', 100, 100, LREAL_TO_DINT(-100*_fDenNum), _stConfig);
TestCaseEncoder('Absolute with Invert 3', -100, -100, LREAL_TO_DINT(100*_fDenNum), _stConfig);

_stConfig.fModulo := 360;
_stConfig.bInvertEncoderDirection := FALSE;
TestCaseEncoder('Modulo 1', 0, 0, LREAL_TO_DINT(0*_fDenNum), _stConfig);
TestCaseEncoder('Modulo 2', 360, 0, LREAL_TO_DINT(0*_fDenNum), _stConfig);
TestCaseEncoder('Modulo 3', 350, 350, LREAL_TO_DINT(350*_fDenNum), _stConfig);
TestCaseEncoder('Modulo 4', -350, -350, LREAL_TO_DINT(-350*_fDenNum), _stConfig);
TestCaseEncoder('Modulo 5', -360, 0, LREAL_TO_DINT(0*_fDenNum), _stConfig);

_stConfig.fModulo := 0;
_stConfig.bInvertEncoderDirection := FALSE;
_stConfig.bIsIntegrator := TRUE;
TestCaseEncoder('Integrate 1', 0, 0, 0, _stConfig);
TestCaseEncoder('Integrate 2', 100, 1, LREAL_TO_DINT(1*_fDenNum), _stConfig);
TestCaseEncoder('Integrate 3', -100, -1, LREAL_TO_DINT(-1*_fDenNum), _stConfig);

_stConfig.fModulo := 0;
_stConfig.bInvertEncoderDirection := FALSE;
_stConfig.bIsIntegrator := FALSE;

_stConfig.fGearFactor := 5;
TestCaseEncoder('GearFactor 1', 0, 0, 0, _stConfig);
TestCaseEncoder('GearFactor 2', 100, 500, LREAL_TO_DINT(500*_fDenNum), _stConfig);
TestCaseEncoder('GearFactor 3', -100, -500, LREAL_TO_DINT(-500*_fDenNum), _stConfig);
_stConfig.fGearFactor := -5;
TestCaseEncoder('GearFactor 4', 100, -500, LREAL_TO_DINT(-500*_fDenNum), _stConfig);
TestCaseEncoder('GearFactor 5', -100, 500, LREAL_TO_DINT(500*_fDenNum), _stConfig);
_stConfig.fGearFactor := 1;

_stConfig.fNumerator := 1E-3;
_stConfig.fDenominator := 2;
_fNumDen := _stConfig.fNumerator / _stConfig.fDenominator;
_fDenNum := _stConfig.fDenominator / _stConfig.fNumerator;

TestCaseEncoder('NumDemFactor 1', 0, 0, LREAL_TO_DINT(0*_fDenNum), _stConfig);
TestCaseEncoder('NumDemFactor 2', 100, 100, LREAL_TO_DINT(100*_fDenNum), _stConfig);
TestCaseEncoder('NumDemFactor 3', -100, -100, LREAL_TO_DINT(-100*_fDenNum), _stConfig);

METHOD TestCase_INC_TO_LREAL
VAR_INPUT
	sName 					: T_MaxString;
	nInput					: DINT;
	fFactor					: LREAL;
	fExpected				: LREAL;
	stConfig				: ST_Encoder_Config;
END_VAR

VAR	
	fbEncoder 				: FB_Encoder;		
	fActual					: LREAL;
	fTolerance 				: REAL := 1E-6;
END_VAR
TEST(sName);

fbEncoder.stConfig := stConfig;

fActual := fbEncoder.INC_TO_LREAL(nInput, fFactor);

AssertEquals_LREAL(Expected := fExpected,
             Actual := fActual,
			 fTolerance,
             Message := 'fResult is not correct');

TEST_FINISHED();
END_METHOD

METHOD TestCase_LREAL_TO_INC
VAR_INPUT
	sName 					: T_MaxString;
	fInput					: LREAL;
	fFactor					: LREAL;
	nExpected				: DINT;
	stConfig				: ST_Encoder_Config;
END_VAR

VAR	
	fbEncoder 				: FB_Encoder;		
	nActual					: DINT;
END_VAR
TEST(sName);

fbEncoder.stConfig := stConfig;

nActual := fbEncoder.LREAL_TO_INC(fInput, fFactor);

AssertEquals_DINT(Expected := nExpected,
             Actual := nActual,
             Message := 'nResult is not correct');	

TEST_FINISHED();
END_METHOD

METHOD TestCaseEncoder
VAR_INPUT
	sName 					: T_MaxString;
	fInput					: REAL;
	fExpected				: LREAL;
	nExpected				: DINT;
	stConfig				: ST_Encoder_Config;
END_VAR

VAR	
	fbEncoder 				: FB_Encoder;
	nCycleCount 			: INT;
	fActual					: LREAL;	
	nActual					: DINT;
	fTolerance 				: REAL := 1E-6;
END_VAR
TEST(sName);

fbEncoder.stConfig := stConfig;
fbEncoder.fValue := fInput;

(*	Call FB to test	*)
FOR nCycleCount := 0 TO 9 DO
   fbEncoder();
END_FOR

(*	Evaluation of results	*)
fActual := fbEncoder.fResult;
nActual := fbEncoder.nResult;

AssertEquals_LREAL(Expected := fExpected,
             Actual := fActual,
			 fTolerance,
             Message := 'fResult is not correct');

AssertEquals_DINT(Expected := nExpected,
             Actual := nActual,
             Message := 'nResult is not correct');	

TEST_FINISHED();
END_METHOD

END_FUNCTION_BLOCK

// ---- Common/Components/Encoder/FB_Encoder.TcPOU
(*
	Generic simulated Encoder 
*)
{attribute 'reflection'} 
FUNCTION_BLOCK FB_Encoder
VAR_INPUT
	fValue 			: LREAL; //Input Value [unit] or [unit/s]	
	stConfig 		: ST_Encoder_Config;	
END_VAR

VAR_OUTPUT
	nResult 		: DINT; //Position [INC]
	fResult 		: LREAL;
END_VAR

VAR
	{attribute 'instance-path'} 
    {attribute 'noinit'} 
    _sPath 				: STRING;
	_fValue 			: LREAL;
END_VAR

InitRun();
ControlLogic();

METHOD PRIVATE ControlLogic
IF stConfig.bIsIntegrator THEN
	_fValue := _fValue + (fValue * stConfig.fGearFactor * GVL_Core.fbSystem.fDeltaTime);
ELSE
	_fValue := fValue * stConfig.fGearFactor;
END_IF

IF stConfig.fModulo > 0.0 THEN
	_fValue := LREAL_TO_REAL(LMOD(_fValue, stConfig.fModulo));
END_IF

fResult := _fValue;

IF stConfig.bInvertEncoderDirection THEN
	nResult := LREAL_TO_INC(fResult, -1);
ELSE
	nResult := LREAL_TO_INC(fResult, 1);	
END_IF
END_METHOD

METHOD INC_TO_LREAL : LREAL
VAR_INPUT
	nValue : DINT;
	fFactor : LREAL;
END_VAR
//Parameters validation
stConfig.fNumerator := MAX(1E-6, stConfig.fNumerator);
stConfig.fDenominator := MAX(1E-6, stConfig.fDenominator);

INC_TO_LREAL := DINT_TO_REAL(nValue) * (stConfig.fNumerator / stConfig.fDenominator) * fFactor;
END_METHOD

METHOD PRIVATE InitRun
VAR_INST
	bInitRun : BOOL := TRUE;
END_VAR
IF NOT bInitRun THEN RETURN; END_IF
bInitRun := FALSE;
END_METHOD

METHOD LREAL_TO_INC : DINT
VAR_INPUT
	fValue : LREAL;
	fFactor : LREAL;
END_VAR
//Parameters validation
stConfig.fNumerator := MAX(1E-6, stConfig.fNumerator);
stConfig.fDenominator := MAX(1E-6, stConfig.fDenominator);

LREAL_TO_INC := LREAL_TO_DINT(fValue * (stConfig.fDenominator / stConfig.fNumerator) * fFactor);
END_METHOD

METHOD PUBLIC SetActualValue : BOOL
VAR_INPUT
	fValue : LREAL;
END_VAR
_fValue := fValue;
END_METHOD

END_FUNCTION_BLOCK

// ---- Common/Components/FB_Clock.TcPOU
FUNCTION_BLOCK FB_Clock
VAR_INPUT
	tPT		: TIME;
END_VAR

VAR_OUTPUT
	bQ		: BOOL;
END_VAR

VAR
	_fbTon1	: TON;
	_fbTon2	: TON;
END_VAR

_fbTon1.PT := tPT;
_fbTon2.PT := tPT;

_fbTon1(IN := NOT bQ);
_fbTon2(IN := bQ);

IF _fbTon1.Q THEN
	bQ := TRUE;
END_IF

IF _fbTon2.Q THEN
	bQ := FALSE;
END_IF

END_FUNCTION_BLOCK

// ---- Common/Components/FB_ClockAdvanced.TcPOU
FUNCTION_BLOCK FB_ClockAdvanced
VAR_INPUT
	bEnable				: BOOL;
	tImpulsePTHigh		: TIME;
	tImpulsePTLow		: TIME;
	tDelay				: TIME;
	bInvert				: BOOL;
END_VAR

VAR_OUTPUT
	bQ					: BOOL;
END_VAR

VAR
	_fbTon1				: TON;
	_fbTon2				: TON;
	_fbTonDelay 		: TON;
	_bValue 			: BOOL;
END_VAR

_fbTonDelay.IN := bEnable;
_fbTonDelay.PT := tDelay;
_fbTonDelay();

IF NOT bEnable THEN
	bQ := FALSE;
	_fbTon1(IN := FALSE);
	_fbTon2(IN := FALSE);
	RETURN;
END_IF

IF _fbTonDelay.Q THEN
	IF bInvert THEN
		_fbTon1.PT := tImpulsePTHigh;
		_fbTon2.PT := tImpulsePTLow;
	ELSE
		_fbTon1.PT := tImpulsePTLow;
		_fbTon2.PT := tImpulsePTHigh;
	END_IF
	
	_fbTon1(IN := NOT _bValue);
	_fbTon2(IN := _bValue);
	
	IF _fbTon1.Q THEN
		_bValue := TRUE;
	END_IF
	
	IF _fbTon2.Q THEN
		_bValue := FALSE;
	END_IF	
	
	IF bInvert THEN
		bQ := NOT _bValue;
	ELSE
		bQ := _bValue;	
	END_IF	
END_IF

END_FUNCTION_BLOCK

// ---- Common/FileIo/FB_FileIO.TcPOU
(*
	File read/write operations.
*)
FUNCTION_BLOCK FB_FileIO
VAR	
	_sNetId				: STRING;
	_fbFileOpen 		: FB_FileOpen;
	_fbFileWrite 		: FB_FileWrite;
	_fbFileRead 		: FB_FileRead;
	_fbFileClose 		: FB_FileClose;	
	_fbCreateDir		: FB_CreateDir;
	_nHFile 			: UINT := 0;
	_eReadState 		: E_FileIoState := READY;
	_eWriteState 		: E_FileIoState := READY;
	_nBytesReadResult	: UDINT;
	_nErrorIdResult		: UDINT;	
END_VAR

(*
	Number of bytes from last read (maps to _nBytesReadResult)
*)
PROPERTY PUBLIC nBytesRead : UDINT
GET
nBytesRead := _nBytesReadResult;
END_GET
SET // PRIVATE
_nBytesReadResult := nBytesRead;
END_SET
END_PROPERTY

(*
	Last error ID (maps to _nErrorIdResult)
*)
PROPERTY PUBLIC nErrorId : uDINT
GET
nErrorId := _nErrorIdResult;
END_GET
SET // PRIVATE
_nErrorIdResult := nErrorId;
END_SET
END_PROPERTY

(*
	Read data from file
	sFileName (T_MaxString): Name/path of the file to read.
	pData (PVOID): Pointer to the data buffer for storing the file contents.
	nLength (UDINT): Number of bytes to read.
*)
METHOD PUBLIC Read : BOOL
VAR_INPUT
	sFileName	: T_MaxString;	//Name/path of the file to read
	pData		: PVOID;	//ointer to the data buffer for storing the file contents
	nLength		: UDINT; //Number of bytes to read
END_VAR
Read := FALSE;
CASE _eReadState OF
	E_FileIoState.READY:
		_fbFileOpen(sNetId := _sNetId, bExecute := FALSE);
		_fbFileRead(sNetId := _sNetId, bExecute := FALSE);
		_fbFileClose(sNetId := _sNetId, bExecute := FALSE);
		_eReadState := E_FileIoState.OPEN;
		
	E_FileIoState.OPEN:
		nErrorId := 0;
		nBytesRead := 0;
		IF _nHFile = 0 THEN
			_fbFileOpen.sPathName := sFileName;
			_fbFileOpen.nMode := FOPEN_MODEREAD;
			_fbFileOpen.ePath := PATH_GENERIC;
			_fbFileOpen(bExecute := TRUE);
		END_IF
		IF _fbFileOpen.hFile <> 0 AND NOT _fbFileOpen.bBusy AND NOT _fbFileOpen.bError THEN
			_nHFile := _fbFileOpen.hFile;
			_fbFileOpen(bExecute := FALSE);			
			_fbFileRead.hFile := _nHFile;
			_fbFileRead.cbReadLen := nLength;
			_fbFileRead.pReadBuff := pData;
			_eReadState := E_FileIoState.READ;
		END_IF
		IF _fbFileOpen.bError THEN
			_fbFileOpen(bExecute := FALSE);
			nErrorId := _fbFileOpen.nErrId;
			_eReadState := E_FileIoState.CREATE;
		END_IF
		
	E_FileIoState.CREATE:
		IF THIS^.Write(sFileName, pData, nLength) THEN
			IF nErrorId = 0 THEN
				_eReadState := E_FileIoState.OPEN;
			ELSE
				_eReadState := E_FileIoState.ERROR;
			END_IF
		END_IF
				
	E_FileIoState.READ:
		_fbFileRead(bExecute := TRUE);
		IF NOT _fbFileRead.bBusy AND NOT _fbFileRead.bError THEN
			nBytesRead := _fbFileRead.cbRead;
			_fbFileRead(bExecute := FALSE);
			_eReadState := E_FileIoState.CLOSE;
		END_IF
		IF _fbFileRead.bError THEN
			nErrorId := _fbFileRead.nErrId;
			_eReadState := E_FileIoState.ERROR;
		END_IF
		
	E_FileIoState.CLOSE:
		IF _nHFile <> 0 THEN
			_fbFileClose(hFile := _nHFile, bExecute := TRUE);
		END_IF
		IF NOT _fbFileClose.bBusy THEN
			_fbFileClose(bExecute := FALSE);
			_nHFile := 0;
			_eReadState := E_FileIoState.READY;
			Read := TRUE;
		END_IF
				
	E_FileIoState.ERROR:
		F_LogError(CONCAT('Error reading/writing file in ', CONCAT(_sNetId, CONCAT(' - ', sFileName))));
		_eReadState := E_FileIoState.CLOSE;
		
END_CASE
END_METHOD

(*
	Network identifier (maps to _sNetId)
*)
PROPERTY sNetId : STRING
GET
sNetId := _sNetId;
END_GET
SET
_sNetId := sNetId;
END_SET
END_PROPERTY

(*
	Write data to file
	sFileName (T_MaxString): Name/path of the file.
	pData (PVOID): Pointer to the content data buffer.
	nLength (UDINT): Number of bytes to write.
*)
METHOD PUBLIC Write : BOOL
VAR_INPUT
	sFileName	: T_MaxString;	//Name/path of the file
	pData 		: PVOID;	//Pointer to the content data buffer
	nLength 	: UDINT;	//Number of bytes to write
END_VAR
Write := FALSE;
CASE _eWriteState OF
	E_FileIoState.READY:
		_fbFileOpen(sNetId := _sNetId, bExecute := FALSE);
		_fbFileWrite(sNetId := _sNetId, bExecute := FALSE);
		_fbFileClose(sNetId := _sNetId, bExecute := FALSE);
		_fbCreateDir(sNetId := _sNetId, bExecute := FALSE);
		_eWriteState := E_FileIoState.OPEN;
		
	E_FileIoState.OPEN:
		nErrorId := 0;
		IF _nHFile = 0 THEN
			_fbFileOpen.sPathName := sFileName;
			_fbFileOpen.nMode := FOPEN_MODEWRITE;
			_fbFileOpen.ePath := PATH_GENERIC;
			_fbFileOpen(bExecute := TRUE);
		END_IF
		IF _fbFileOpen.hFile <> 0 AND NOT _fbFileOpen.bBusy AND NOT _fbFileOpen.bError THEN
			_nHFile := _fbFileOpen.hFile;
			_fbFileOpen(bExecute := FALSE);					
			_fbFileWrite.hFile := _nHFile;
			_fbFileWrite.cbWriteLen := nLength;
			_fbFileWrite.pWriteBuff := pData;
			_eWriteState := E_FileIoState.WRITE;
		END_IF
		IF _fbFileOpen.bError THEN
			_fbFileOpen(bExecute := FALSE);
			nErrorId := _fbFileOpen.nErrId;
			_eWriteState := E_FileIoState.CREATE;			
		END_IF
		
	E_FileIoState.CREATE:
		_fbCreateDir.sPathName:= sFileName;
		_fbCreateDir.ePath:= PATH_GENERIC;
		_fbCreateDir(bExecute := TRUE);
		IF NOT _fbCreateDir.bBusy AND NOT _fbCreateDir.bError THEN
			nErrorId := 0;
			_fbCreateDir(bExecute := FALSE);
			_eWriteState := E_FileIoState.OPEN;
		END_IF
		IF _fbCreateDir.bError THEN
			nErrorId := _fbCreateDir.nErrId;
			_eWriteState := E_FileIoState.ERROR;			
		END_IF
				
	E_FileIoState.WRITE:
		_fbFileWrite(bExecute := TRUE);
		IF NOT _fbFileWrite.bBusy AND _fbFileWrite.cbWrite = nLength AND NOT _fbFileWrite.bError THEN
			_fbFileWrite(bExecute := FALSE);
			_eWriteState := E_FileIoState.CLOSE;
		END_IF
		IF _fbFileWrite.bError THEN
			nErrorId := _fbFileWrite.nErrId;
			_eWriteState := E_FileIoState.ERROR;
		END_IF
		
	E_FileIoState.CLOSE:
		IF  _nHFile <> 0 THEN
			_fbFileClose(hFile := _nHFile, bExecute := TRUE);
		END_IF
		IF NOT _fbFileClose.bBusy THEN
			_fbFileClose(bExecute := FALSE);
			_nHFile := 0;
			_eWriteState := E_FileIoState.READY;
			Write := TRUE;
		END_IF

	E_FileIoState.ERROR:
		F_LogError(CONCAT('Error reading/writing file in ', CONCAT(_sNetId, CONCAT(' - ', sFileName))));
		_eWriteState := E_FileIoState.CLOSE;	

END_CASE
END_METHOD

END_FUNCTION_BLOCK
